{attribute 'qualified_only'}
{attribute 'strict'}
{attribute 'to_string'}
TYPE E_StateDoorCtrl :
(
	NotReady,
	DoorClosed ,
	DoorOpening ,
	DoorOpen , // hier wird dann einfach zahl 2 hinterlegt
	DoorClosing ,
	Error := 90);
// eStateDoorCtrl := UINT;
END_TYPE

(* stored: Version 1.1.0.1
   DUT E_StateDoorCtrl: Id {92cbf0b1-afb1-434d-9e08-9c9f741242d4} *)
